// TIA Portal V19 export
TYPE "type_cmParError"
// stored: Access Published
   STRUCT
      error : Bool;
   END_STRUCT;
END_TYPE
